PROGRAM MAIN
VAR
END_VAR

END_PROGRAM

(* stored: Version 1.1.0.1
   POU MAIN: Id {8710c1e6-9a0c-4c98-b38a-50b05c98f6e7} *)
